FUNCTION_BLOCK Station_Status (* Basic Function Block Type *)
  (* Standard: 61499-2 *)
  (* Version 0.0, 7/18/2025, Evans_A, Schneider Electric, Template *)
  PACKAGE Main;
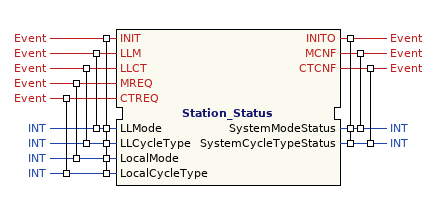
  EVENT_INPUT
    INIT WITH LLMode, LLCycleType, LocalMode, LocalCycleType; (* Initialization Request *)
    LLM WITH LLMode; (* Normal Execution Request *)
    LLCT WITH LLCycleType;
    MREQ WITH LocalMode;
    CTREQ WITH LocalCycleType;
  END_EVENT
  EVENT_OUTPUT
    INITO WITH SystemModeStatus, SystemCycleTypeStatus; (* Initialization Confirm *)
    MCNF WITH SystemModeStatus; (* Execution Confirmation *)
    CTCNF WITH SystemCycleTypeStatus;
  END_EVENT
  VAR_INPUT
    LLMode : INT; (* Input event qualifier *)
    LLCycleType : INT;
    LocalMode : INT;
    LocalCycleType : INT;
  END_VAR
  VAR_OUTPUT
    SystemModeStatus : INT; (* Output event qualifier *)
    SystemCycleTypeStatus : INT;
  END_VAR
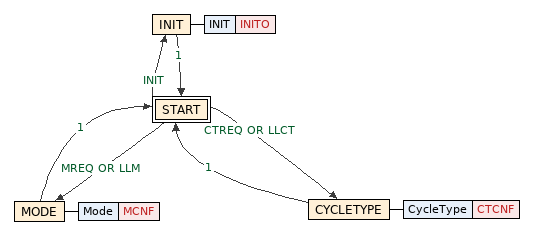
  EC_STATES
    START; (* Initial State *)
    INIT : INIT -> INITO; (* Initialization *)
    MODE : Mode -> MCNF; (* Normal execution *)
    CYCLETYPE : CycleType -> CTCNF;
  END_STATES
  EC_TRANSITIONS
    START TO INIT := INIT;
    INIT TO START := 1;
    START TO MODE := MREQ OR LLM;
    MODE TO START := 1;
    START TO CYCLETYPE := CTREQ OR LLCT;
    CYCLETYPE TO START := 1;
  END_TRANSITIONS
  ALGORITHM INIT IN ST: (* Initialization algorithm *)
;
  END_ALGORITHM
  ALGORITHM Mode IN ST: (* Normally executed algorithm *)
IF LLMode = LocalMode THEN
	SystemModeStatus := LocalMode;
ELSE
	SystemModeStatus := 100;
END_IF;
  END_ALGORITHM
  ALGORITHM CycleType IN ST:
IF LLCycleType = LocalCycleType THEN
	SystemCycleTypeStatus := LocalCycleType;
ELSE
	SystemCycleTypeStatus := 100;
END_IF;
  END_ALGORITHM
END_FUNCTION_BLOCK
